PROGRAM POU_Manual_Auto
VAR
END_VAR

// NETWORK 1

END_PROGRAM

(* stored: Version 1.1.0.1, ProductVersion 3.1.4024.0
   POU POU_Manual_Auto: Id {daa6effe-2521-4ee6-890a-c3171add926d}, SpecialFunc None *)
